TYPE BinaryAssertionsStructure :
STRUCT
	
	
END_STRUCT
END_TYPE

(* stored: Version 1.1.0.1, ProductVersion 3.1.4024.11
   DUT BinaryAssertionsStructure: Id {51357290-15f0-4fa8-bb61-bba7d77481cf} *)
